{attribute 'qualified_only'}
VAR_GLOBAL
	Lh_in:BOOL;
	Lh_out:BOOL;
	Rh_in:BOOL;
	Rh_out:BOOL;
	Single_drum:BOOL;
END_VAR

(* stored: Version 1.1.0.1, ProductVersion 3.1.4024.0
   GVL Clutch: Id {a0bd0f36-a135-4ad8-9939-5693397818bb} *)
